// TIA Portal project "TRFİKK" (V16)

(* hardware
DEVICE "S7-1200 station_1"  S7-1200 Station
   slot 0: "Rack_0"  S7-1200 Rack  Rack  V1.0
   slot 1: "PLC_1"  CPU 1212C DC/DC/Rly  6ES7 212-1HE40-0XB0  V4.4
   slot 2: "DI 8x24VDC_1"  6ES7 221-1BF32-0XB0  V2.0
   slot 3: "DQ 8x24VDC _1"  SM 1222 DQ8 x 24VDC  6ES7 222-1BF32-0XB0  V2.0
   slot 3: "DQ 4x5VDC_1"  DQ4 signal board (200 kHz)  6ES7 222-1AD30-0XB0  V1.0
*)

// ===== PLC "PLC_1"  CPU 1212C DC/DC/Rly =====

VAR_GLOBAL   // PLC tag table "Default tag table"
   "Clock_Byte" AT %MB0 : Byte;
   "Clock_10Hz" AT %M0.0 : Bool;
   "Clock_5Hz" AT %M0.1 : Bool;
   "Clock_2.5Hz" AT %M0.2 : Bool;
   "Clock_2Hz" AT %M0.3 : Bool;
   "Clock_1.25Hz" AT %M0.4 : Bool;
   "Clock_1Hz" AT %M0.5 : Bool;
   "Clock_0.625Hz" AT %M0.6 : Bool;
   "Clock_0.5Hz" AT %M0.7 : Bool;
   "start but" AT %I0.0 : Bool;
   "stop but" AT %I0.1 : Bool;
   "gece sistem but" AT %I0.2 : Bool;
   "gece sistem stop but" AT %I0.3 : Bool;
   "1. yaya but" AT %I0.4 : Bool;
   "2. yaya but" AT %I0.5 : Bool;
   "3.yaya but" AT %I0.6 : Bool;
   "4. yaya but" AT %I0.7 : Bool;
   "5.yaya but" AT %I8.0 : Bool;
   "6.yaya but" AT %I8.1 : Bool;
   "7.yaya but" AT %I8.2 : Bool;
   "8.yaya but" AT %I8.3 : Bool;
   "kırmızı1" AT %Q0.0 : Bool;
   "sarı1" AT %Q0.1 : Bool;
   "yeşil1" AT %Q0.2 : Bool;
   "kırmızı2" AT %Q0.3 : Bool;
   "sarı2" AT %Q0.4 : Bool;
   "yeşil2" AT %Q0.5 : Bool;
   "kırmızı3" AT %Q12.0 : Bool;
   "sarı3" AT %Q12.1 : Bool;
   "yeşil3" AT %Q12.2 : Bool;
   "kırmızı4" AT %Q12.3 : Bool;
   "sarı4" AT %Q12.4 : Bool;
   "yeşil4" AT %Q12.5 : Bool;
   "start mem" AT %M10.0 : Bool;
   "gece sis mem" AT %M10.1 : Bool;
   "Tag_1" AT %M10.2 : Bool;
   "Tag_2" AT %M10.3 : Bool;
   "GECE LAMBA SENSÖR" AT %I8.4 : Bool;
   "1.CADDE LAMBA" AT %M50.0 : Bool;
   "2. CADDE LAMBA" AT %M50.1 : Bool;
   "3. CADDE İÇİN LAMBA" AT %M50.2 : Bool;
   "4. CADDE LAMBA" AT %M50.3 : Bool;
   "yayahafıza but" AT %M60.0 : Bool;
   "YAYAHAFIZABUTON" AT %M60.1 : Bool;
   "kırmızı5" AT %Q12.6 : Bool;
   "sarı5" AT %Q12.7 : Bool;
   "yeşil5" AT %Q4.0 : Bool;
   "kırmızı6" AT %Q4.1 : Bool;
   "sarı6" AT %Q4.2 : Bool;
   "yeşil6" AT %Q4.3 : Bool;
END_VAR

// folder: System blocks/Program resources

DATA_BLOCK "timer1"   // DB1
{ S7_Optimized_Access := 'TRUE' }
AUTHOR : Simatic
FAMILY : IEC
NAME : IEC_TMR
VERSION : 1.0
// stored: InstanceOfName IEC_TIMER
"IEC_TIMER"
BEGIN
END_DATA_BLOCK

DATA_BLOCK "timer7"   // DB4
{ S7_Optimized_Access := 'TRUE' }
AUTHOR : Simatic
FAMILY : IEC
NAME : IEC_TMR
VERSION : 1.0
// stored: InstanceOfName IEC_TIMER
"IEC_TIMER"
BEGIN
END_DATA_BLOCK

DATA_BLOCK "TİMER10"   // DB6
{ S7_Optimized_Access := 'TRUE' }
AUTHOR : Simatic
FAMILY : IEC
NAME : IEC_TMR
VERSION : 1.0
// stored: InstanceOfName IEC_TIMER
"IEC_TIMER"
BEGIN
END_DATA_BLOCK

// folder: (top level)

FUNCTION "Block_1" : Void   // FC1, LAD
{ S7_Optimized_Access := 'TRUE' }
VERSION : 0.1
BEGIN

REGION Network 1
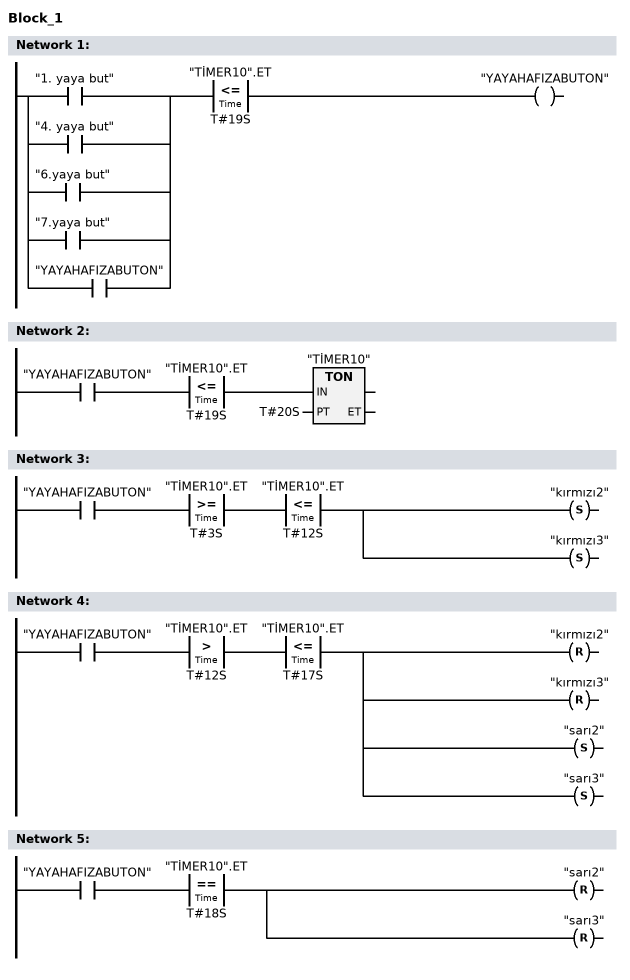
   RUNG wire#powerrail
      Contact( "1. yaya but" )
      wire#w1
      { S7_Templates := "SrcType := Time" } LE_Contact(in1 := "TİMER10".ET, in2 := T#19S)
      Coil( "YAYAHAFIZABUTON" )
   END_RUNG
   RUNG wire#powerrail
      Contact( "4. yaya but" )
   END_RUNG wire#w1
   RUNG wire#powerrail
      Contact( "6.yaya but" )
   END_RUNG wire#w1
   RUNG wire#powerrail
      Contact( "7.yaya but" )
   END_RUNG wire#w1
   RUNG wire#powerrail
      Contact( "YAYAHAFIZABUTON" )
   END_RUNG wire#w1
   // the same network as SCL:
   "YAYAHAFIZABUTON" := ("1. yaya but" OR "4. yaya but" OR "6.yaya but" OR "7.yaya but" OR "YAYAHAFIZABUTON") AND ("TİMER10".ET <= T#19S);
END_REGION

REGION Network 2
   "TİMER10".TON(IN := "YAYAHAFIZABUTON" AND ("TİMER10".ET <= T#19S), PT := T#20S);
END_REGION

REGION Network 3
   RUNG wire#powerrail
      Contact( "YAYAHAFIZABUTON" )
      { S7_Templates := "SrcType := Time" } GE_Contact(in1 := "TİMER10".ET, in2 := T#3S)
      { S7_Templates := "SrcType := Time" } LE_Contact(in1 := "TİMER10".ET, in2 := T#12S)
      wire#w1
      S_Coil( "kırmızı2" )
   END_RUNG
   RUNG wire#w1
      S_Coil( "kırmızı3" )
   END_RUNG
   // the same network as SCL:
   IF "YAYAHAFIZABUTON" AND ("TİMER10".ET >= T#3S) AND ("TİMER10".ET <= T#12S) THEN
       "kırmızı2" := TRUE;
       "kırmızı3" := TRUE;
   END_IF;
END_REGION

REGION Network 4
   RUNG wire#powerrail
      Contact( "YAYAHAFIZABUTON" )
      { S7_Templates := "SrcType := Time" } GT_Contact(in1 := "TİMER10".ET, in2 := T#12S)
      { S7_Templates := "SrcType := Time" } LE_Contact(in1 := "TİMER10".ET, in2 := T#17S)
      wire#w1
      R_Coil( "kırmızı2" )
   END_RUNG
   RUNG wire#w1
      R_Coil( "kırmızı3" )
   END_RUNG
   RUNG wire#w1
      S_Coil( "sarı2" )
   END_RUNG
   RUNG wire#w1
      S_Coil( "sarı3" )
   END_RUNG
   // the same network as SCL:
   IF "YAYAHAFIZABUTON" AND ("TİMER10".ET > T#12S) AND ("TİMER10".ET <= T#17S) THEN
       "kırmızı2" := FALSE;
       "kırmızı3" := FALSE;
       "sarı2" := TRUE;
       "sarı3" := TRUE;
   END_IF;
END_REGION

REGION Network 5
   RUNG wire#powerrail
      Contact( "YAYAHAFIZABUTON" )
      { S7_Templates := "SrcType := Time" } EQ_Contact(in1 := "TİMER10".ET, in2 := T#18S)
      wire#w1
      R_Coil( "sarı2" )
   END_RUNG
   RUNG wire#w1
      R_Coil( "sarı3" )
   END_RUNG
   // the same network as SCL:
   IF "YAYAHAFIZABUTON" AND ("TİMER10".ET = T#18S) THEN
       "sarı2" := FALSE;
       "sarı3" := FALSE;
   END_IF;
END_REGION
END_FUNCTION

ORGANIZATION_BLOCK "Main"   // OB1, LAD, ProgramCycle
TITLE = "Main Program Sweep (Cycle)"
{ S7_Optimized_Access := 'TRUE' }
VERSION : 0.1
   VAR_INPUT
      Initial_Call : Bool;   // Initial call of this OB
      Remanence : Bool;   // =True, if remanent data are available
   END_VAR
   VAR_TEMP   // added for the SCL form of the ladder/FBD networks
      _w1 : Bool;
   END_VAR
BEGIN

REGION Network 1: sistem start memory
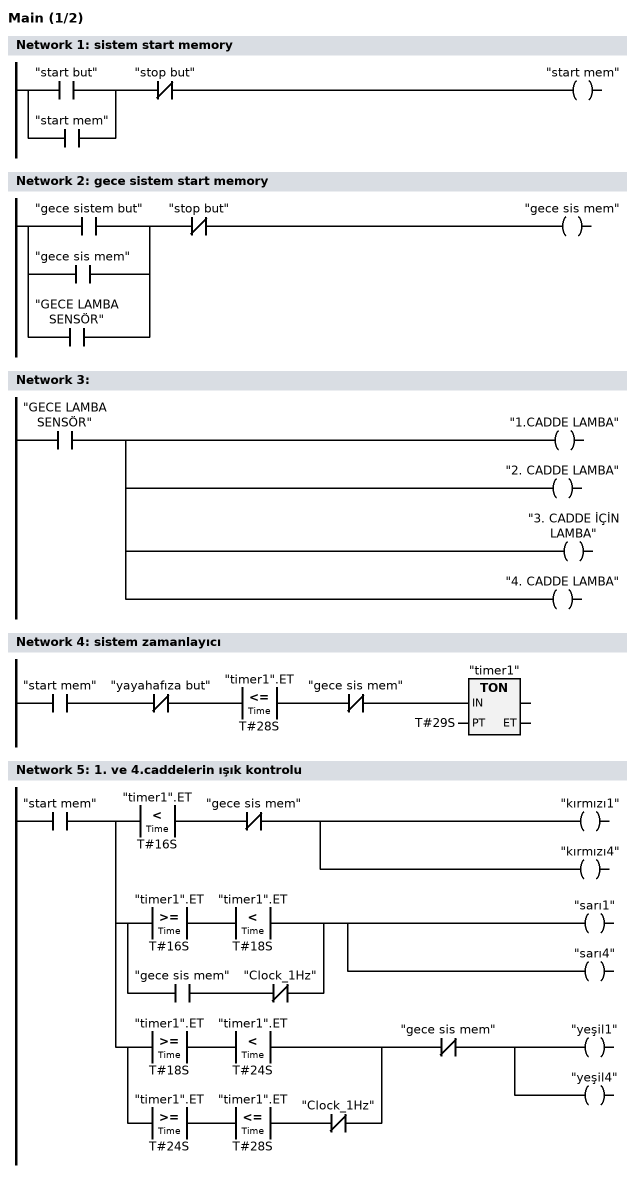
   RUNG wire#powerrail
      Contact( "start but" )
      wire#w1
      I_Contact( "stop but" )
      Coil( "start mem" )
   END_RUNG
   RUNG wire#powerrail
      Contact( "start mem" )
   END_RUNG wire#w1
   // the same network as SCL:
   "start mem" := ("start but" OR "start mem") AND NOT "stop but";
END_REGION

REGION Network 2: gece sistem start memory
   RUNG wire#powerrail
      Contact( "gece sistem but" )
      wire#w1
      I_Contact( "stop but" )
      Coil( "gece sis mem" )
   END_RUNG
   RUNG wire#powerrail
      Contact( "gece sis mem" )
   END_RUNG wire#w1
   RUNG wire#powerrail
      Contact( "GECE LAMBA SENSÖR" )
   END_RUNG wire#w1
   // the same network as SCL:
   "gece sis mem" := ("gece sistem but" OR "gece sis mem" OR "GECE LAMBA SENSÖR") AND NOT "stop but";
END_REGION

REGION Network 3
   RUNG wire#powerrail
      Contact( "GECE LAMBA SENSÖR" )
      wire#w1
      Coil( "1.CADDE LAMBA" )
   END_RUNG
   RUNG wire#w1
      Coil( "2. CADDE LAMBA" )
   END_RUNG
   RUNG wire#w1
      Coil( "3. CADDE İÇİN LAMBA" )
   END_RUNG
   RUNG wire#w1
      Coil( "4. CADDE LAMBA" )
   END_RUNG
   // the same network as SCL:
   "1.CADDE LAMBA" := "GECE LAMBA SENSÖR";
   "2. CADDE LAMBA" := "GECE LAMBA SENSÖR";
   "3. CADDE İÇİN LAMBA" := "GECE LAMBA SENSÖR";
   "4. CADDE LAMBA" := "GECE LAMBA SENSÖR";
END_REGION

REGION Network 4: sistem zamanlayıcı
   "timer1".TON(IN := "start mem" AND NOT "yayahafıza but" AND ("timer1".ET <= T#28S) AND NOT "gece sis mem",
                PT := T#29S);
END_REGION

REGION Network 5: 1. ve 4.caddelerin ışık kontrolu
   RUNG wire#powerrail
      Contact( "start mem" )
      wire#w1
      { S7_Templates := "SrcType := Time" } LT_Contact(in1 := "timer1".ET, in2 := T#16S)
      I_Contact( "gece sis mem" )
      wire#w2
      Coil( "kırmızı1" )
   END_RUNG
   RUNG wire#w2
      Coil( "kırmızı4" )
   END_RUNG
   RUNG wire#w1
      { S7_Templates := "SrcType := Time" } GE_Contact(in1 := "timer1".ET, in2 := T#16S)
      { S7_Templates := "SrcType := Time" } LT_Contact(in1 := "timer1".ET, in2 := T#18S)
      wire#w3
      Coil( "sarı1" )
   END_RUNG
   RUNG wire#w1
      Contact( "gece sis mem" )
      I_Contact( "Clock_1Hz" )
   END_RUNG wire#w3
   RUNG wire#w3
      Coil( "sarı4" )
   END_RUNG
   RUNG wire#w1
      { S7_Templates := "SrcType := Time" } GE_Contact(in1 := "timer1".ET, in2 := T#18S)
      { S7_Templates := "SrcType := Time" } LT_Contact(in1 := "timer1".ET, in2 := T#24S)
      wire#w4
      I_Contact( "gece sis mem" )
      wire#w5
      Coil( "yeşil1" )
   END_RUNG
   RUNG wire#w1
      { S7_Templates := "SrcType := Time" } GE_Contact(in1 := "timer1".ET, in2 := T#24S)
      { S7_Templates := "SrcType := Time" } LE_Contact(in1 := "timer1".ET, in2 := T#28S)
      I_Contact( "Clock_1Hz" )
   END_RUNG wire#w4
   RUNG wire#w5
      Coil( "yeşil4" )
   END_RUNG
   // the same network as SCL:
   "kırmızı1" := "start mem" AND ("timer1".ET < T#16S) AND NOT "gece sis mem";
   "kırmızı4" := "kırmızı1";
   "sarı1" := "start mem" AND ((("timer1".ET >= T#16S) AND ("timer1".ET < T#18S)) OR ("gece sis mem" AND NOT "Clock_1Hz"));
   "sarı4" := "sarı1";
   "yeşil1" := "start mem" AND ((("timer1".ET >= T#18S) AND ("timer1".ET < T#24S)) OR (("timer1".ET >= T#24S) AND ("timer1".ET <= T#28S) AND NOT "Clock_1Hz")) AND NOT "gece sis mem";
   "yeşil4" := "yeşil1";
END_REGION

REGION Network 6: 2. ve 3. caddelerin ışık kontrolu
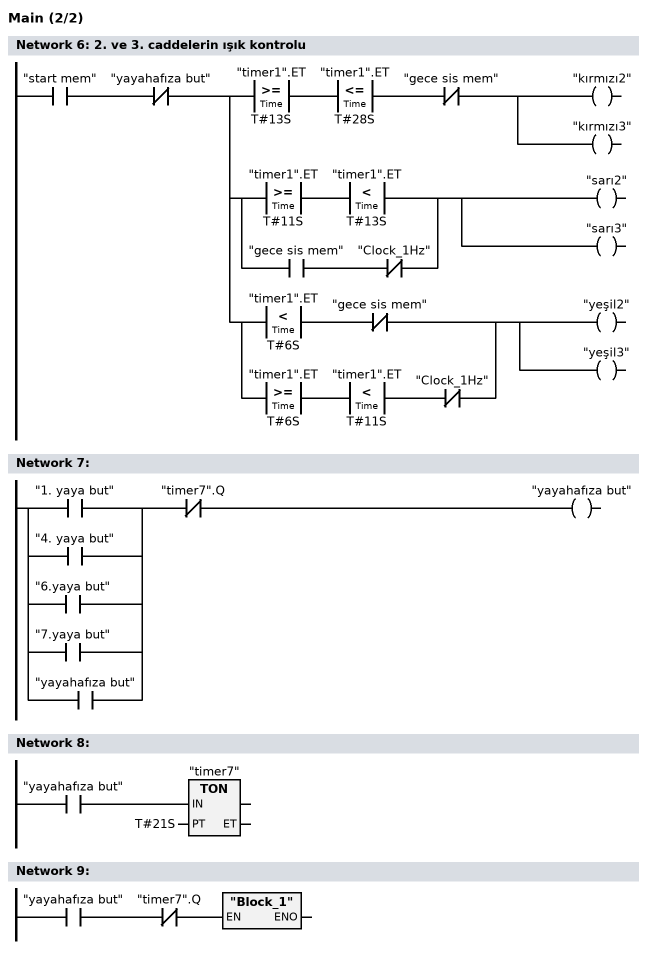
   RUNG wire#powerrail
      Contact( "start mem" )
      I_Contact( "yayahafıza but" )
      wire#w1
      { S7_Templates := "SrcType := Time" } GE_Contact(in1 := "timer1".ET, in2 := T#13S)
      { S7_Templates := "SrcType := Time" } LE_Contact(in1 := "timer1".ET, in2 := T#28S)
      I_Contact( "gece sis mem" )
      wire#w2
      Coil( "kırmızı2" )
   END_RUNG
   RUNG wire#w2
      Coil( "kırmızı3" )
   END_RUNG
   RUNG wire#w1
      { S7_Templates := "SrcType := Time" } GE_Contact(in1 := "timer1".ET, in2 := T#11S)
      { S7_Templates := "SrcType := Time" } LT_Contact(in1 := "timer1".ET, in2 := T#13S)
      wire#w3
      Coil( "sarı2" )
   END_RUNG
   RUNG wire#w1
      Contact( "gece sis mem" )
      I_Contact( "Clock_1Hz" )
   END_RUNG wire#w3
   RUNG wire#w3
      Coil( "sarı3" )
   END_RUNG
   RUNG wire#w1
      { S7_Templates := "SrcType := Time" } LT_Contact(in1 := "timer1".ET, in2 := T#6S)
      I_Contact( "gece sis mem" )
      wire#w4
      Coil( "yeşil2" )
   END_RUNG
   RUNG wire#w1
      { S7_Templates := "SrcType := Time" } GE_Contact(in1 := "timer1".ET, in2 := T#6S)
      { S7_Templates := "SrcType := Time" } LT_Contact(in1 := "timer1".ET, in2 := T#11S)
      I_Contact( "Clock_1Hz" )
   END_RUNG wire#w4
   RUNG wire#w4
      Coil( "yeşil3" )
   END_RUNG
   // the same network as SCL:
   #_w1 := "start mem" AND NOT "yayahafıza but";
   "kırmızı2" := #_w1 AND ("timer1".ET >= T#13S) AND ("timer1".ET <= T#28S) AND NOT "gece sis mem";
   "kırmızı3" := "kırmızı2";
   "sarı2" := #_w1 AND ((("timer1".ET >= T#11S) AND ("timer1".ET < T#13S)) OR ("gece sis mem" AND NOT "Clock_1Hz"));
   "sarı3" := "sarı2";
   "yeşil2" := #_w1 AND ((("timer1".ET < T#6S) AND NOT "gece sis mem") OR (("timer1".ET >= T#6S) AND ("timer1".ET < T#11S) AND NOT "Clock_1Hz"));
   "yeşil3" := "yeşil2";
END_REGION

REGION Network 7
   RUNG wire#powerrail
      Contact( "1. yaya but" )
      wire#w1
      I_Contact( "timer7".Q )
      Coil( "yayahafıza but" )
   END_RUNG
   RUNG wire#powerrail
      Contact( "4. yaya but" )
   END_RUNG wire#w1
   RUNG wire#powerrail
      Contact( "6.yaya but" )
   END_RUNG wire#w1
   RUNG wire#powerrail
      Contact( "7.yaya but" )
   END_RUNG wire#w1
   RUNG wire#powerrail
      Contact( "yayahafıza but" )
   END_RUNG wire#w1
   // the same network as SCL:
   "yayahafıza but" := ("1. yaya but" OR "4. yaya but" OR "6.yaya but" OR "7.yaya but" OR "yayahafıza but") AND NOT "timer7".Q;
END_REGION

REGION Network 8
   "timer7".TON(IN := "yayahafıza but", PT := T#21S);
END_REGION

REGION Network 9
   RUNG wire#powerrail
      Contact( "yayahafıza but" )
      I_Contact( "timer7".Q )
      "Block_1"()
   END_RUNG
   // the same network as SCL:
   IF "yayahafıza but" AND NOT "timer7".Q THEN "Block_1"(); END_IF;
END_REGION
END_ORGANIZATION_BLOCK